FUNCTION_BLOCK FB2_Control
VAR_INPUT
END_VAR
VAR_OUTPUT
END_VAR
VAR
END_VAR

//loadingstation
Parts.Loadingstation(i_inputbelt := Parts.Belt.q_BoxReady, 
	iq_Commandstate := Parts.GlobalCommandState,
	i_weighbridge := Parts.Weighbridge.q_Output,
	q_crane => Parts.Crane.i_Input.AllowedToOperate);

END_FUNCTION_BLOCK

(* stored: Version 1.1.0.1, ProductVersion 3.1.4024.6
   POU FB2_Control: Id {f3ae371c-7e7d-41b3-b42c-11221479fa8f}, SpecialFunc None *)
